// TwinCAT 3 PLC project Untitled1
// ProgramVersion: 3.1.0.9
// libraries:
//   Standard, * (System)
//   VisuElem3DPath, 3.5.6.0 (System)
//   VisuElemMeter, 3.5.6.0 (System)
//   VisuElems, 3.5.6.10 (System)
//   VisuElemsDateTime, 3.5.6.0 (System)
//   VisuElemsSpecialControls, 3.5.6.0 (System)
//   VisuElemsWinControls, 3.5.6.0 (System)
//   VisuElemTextEditor, 3.5.6.0 (System)
//   visuinputs, 3.5.6.0 (system)
//   VisuNativeControl, 3.5.6.0 (System)
//   Tc2_Standard, * (Beckhoff Automation GmbH)
//   Tc2_System, * (Beckhoff Automation GmbH)
//   Tc3_Interfaces, * (Beckhoff Automation GmbH)
//   Tc3_Module, * (Beckhoff Automation GmbH)
// project tree:
//   / GlobalTextList.TcGTLO, PlcTask.TcTTO, Visualization Manager.TcVMO (not stored)
//   POUs/ LADDER1.TcPOU, MAIN.TcPOU
//   VISUs/ Visualization.TcVIS
// real-time tasks:
//   TASK PlcTask: cycle T#10ms, priority 20, ADS port 350

CONFIGURATION Untitled1
    RESOURCE PLC ON TwinCAT3
        TASK PlcTask(INTERVAL := T#10ms, PRIORITY := 20);
        PROGRAM MAIN WITH PlcTask : MAIN;
    END_RESOURCE
END_CONFIGURATION

// ---- POUs/MAIN.TcPOU
PROGRAM MAIN
VAR
END_VAR

LADDER1();

END_PROGRAM

// ---- POUs/LADDER1.TcPOU
PROGRAM LADDER1
VAR
	stop: BOOL;
	start: BOOL;
	emergency: BOOL;
	S_place: BOOL;
	S_full: BOOL;
	S_empty: BOOL;
	S_loading: BOOL;
	S_unload: BOOL;
	valve: BOOL;
	Motor: BOOL;
	y1: BOOL;
	y3: BOOL;
	y2:BOOL;
	TankEmpty: BOOL;
    CU: BOOL; 
    RESET: BOOL; 
    PV: WORD; 
	FILLING: BOOL;
	CV: WORD;
	Q: Bool;
	counter: CTU;
END_VAR
VAR // added by the converter: edge detectors and wires of the graphical bodies
    _w1, _w2 : BOOL;
END_VAR

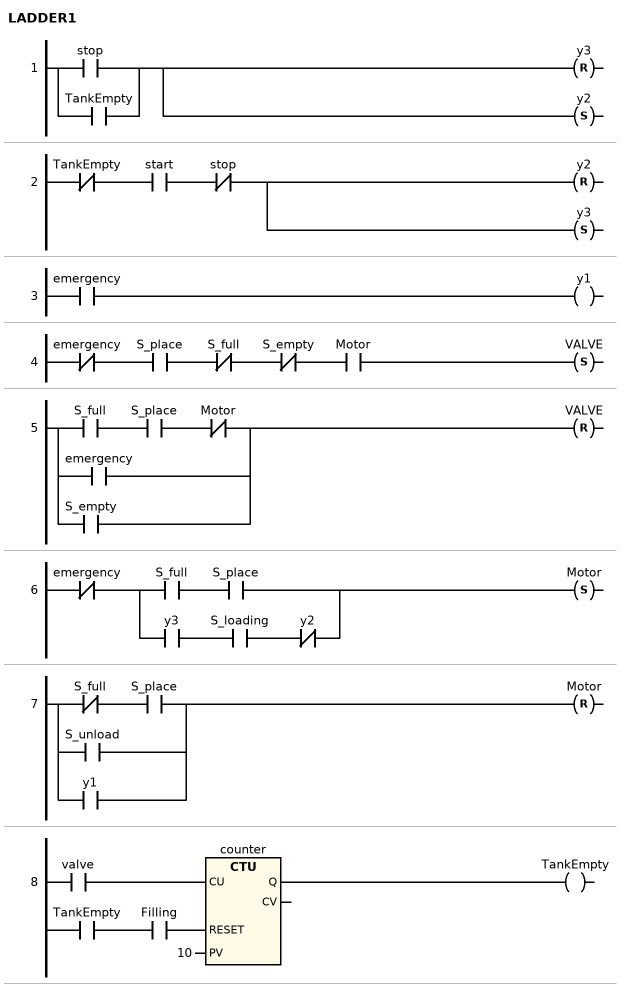
// NETWORK 1
_w1 := stop OR TankEmpty;
y3 R= _w1;
y2 S= _w1;

// NETWORK 2
_w2 := NOT TankEmpty AND start AND NOT stop;
y2 R= _w2;
y3 S= _w2;

// NETWORK 3
y1 := emergency;

// NETWORK 4
VALVE S= NOT emergency AND S_place AND NOT S_full AND NOT S_empty AND Motor;

// NETWORK 5
VALVE R= S_full AND S_place AND NOT Motor OR emergency OR S_empty;

// NETWORK 6
Motor S= NOT emergency AND (S_full AND S_place OR y3 AND S_loading AND NOT y2);

// NETWORK 7
Motor R= NOT S_full AND S_place OR S_unload OR y1;

// NETWORK 8
counter(CU := valve, RESET := TankEmpty AND Filling, PV := 10); // CTU
TankEmpty := counter.Q;

END_PROGRAM

// ---- GlobalTextList.TcGTLO
TEXTLIST GlobalTextList
  16 = 'CONTAINER FULL'
  17 = 'CONTAINER IN PLACE'
  22 = 'Counter : '
  23 = 'Counter : %d'
  24 = 'Counter : %i'
  21 = 'Counter : %s'
  2 = 'emergency'
  25 = 'Emergency Stop'
  26 = 'EMERGENCY STOP'
  13 = 'Filling'
  14 = 'LOADING'
  8 = 'Motor'
  18 = 'MOTOR'
  5 = 'S-empty'
  4 = 'S-full'
  6 = 'S-loading'
  3 = 'S-place'
  7 = 'S-unload'
  0 = 'start'
  1 = 'stop'
  11 = 'S_load'
  12 = 'S_loading'
  19 = 'TANK EMPTY'
  10 = 'tank-empty'
  15 = 'UNLOADING'
  9 = 'valve'
  20 = 'VALVE'
END_TEXTLIST

// ---- VISUs/Visualization.TcVIS
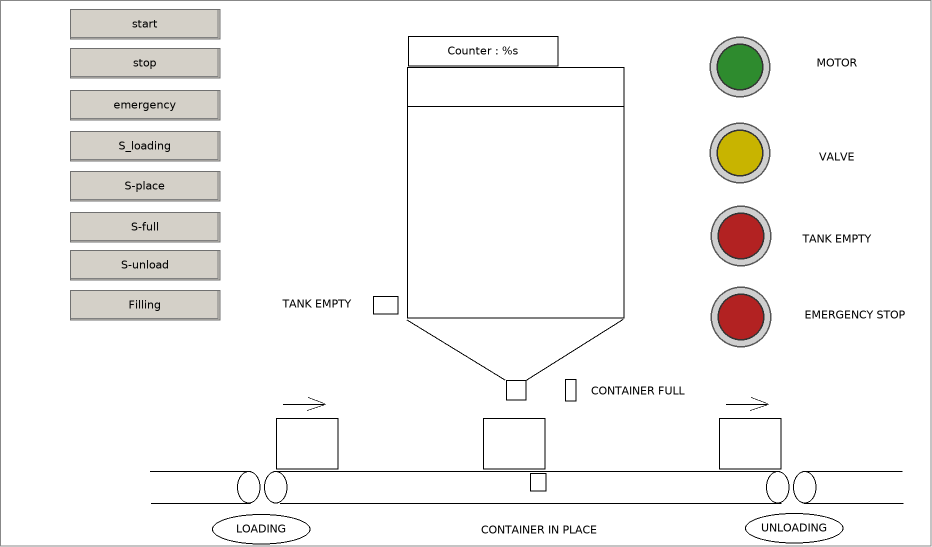
VISUALIZATION Visualization  // 932x547
    Lamp1 (705,32 70x70), variable: LADDER1.Motor, style: Lamp-Lamp1-Green
    Button (70,9 150x30), "start"
        OnMouseDown: toggle LADDER1.start
    Button (70,48 150x30), "stop"
        OnMouseDown: toggle LADDER1.stop
    Button (70,212 150x30), "S-full"
        OnMouseDown: toggle LADDER1.S_full
    Button (70,171 150x30), "S-place"
        OnMouseDown: toggle LADDER1.S_place
    Button (70,90 150x30), "emergency"
        OnMouseDown: toggle LADDER1.emergency
    Lamp1 (705,118 70x70), variable: LADDER1.valve, style: Lamp-Lamp1-Yellow
    Lamp1 (706,201 70x70), variable: LADDER1.TankEmpty, style: Lamp-Lamp1-Red
    Button (70,250 150x30), "S-unload"
        OnMouseDown: toggle LADDER1.S_unload
    Button (70,131 150x30), "S_loading"
        OnMouseDown: toggle LADDER1.S_loading
    Button (70,290 150x30), "Filling"
        OnMouseDown: toggle LADDER1.FILLING
    Rectangle (407,67 217x251)
    Rectangle (407,106 217x212), invisible if: LADDER1.TankEmpty
    Line (413,321)
    Line (505,380) (407,320)
    Line (585,354)
    Line (526,380) (623,319)
    Rectangle (506,380 20x20)
    Rectangle (483,418 62x51), colour toggle: LADDER1.S_full
        OnMouseDown: toggle LADDER1.S_full
    Rectangle (276,418 62x51)
    Rectangle (719,418 62x51)
    Line (726,404) (767,404)
    Line (751,397) (767,403)
    Line (750,410) (768,404)
    Line (283,404) (324,404)
    Line (308,397) (324,403)
    Line (307,410) (325,404)
    Ellipse (264,471 23x32)
    Line (278,471) (779,471)
    Ellipse (766,471 23x32)
    Line (280,503) (781,503)
    Ellipse (237,471 23x32)
    Ellipse (793,471 23x32)
    Line (803,471) (902,471)
    Line (804,503) (903,503)
    Line (150,471) (249,471)
    Line (151,503) (250,503)
    Ellipse (212,514 98x30), "LOADING"
    Ellipse (745,513 98x30), "UNLOADING"
    Rectangle (530,473 16x18)
    Rectangle (565,379 11x22)
    Label (549,376 178x30), "CONTAINER FULL"
    Label (464,515 150x30), "CONTAINER IN PLACE"
    Label (750,42 174x42), "MOTOR"
    Label (750,136 174x42), "VALVE"
    Label (750,218 174x42), "TANK EMPTY"
    Label (242,289 150x30), "TANK EMPTY"
    Rectangle (373,296 25x18)
    Rectangle (408,36 150x30), "Counter : %s", text variable: MAIN.LADDER1.counter.CV
    Lamp1 (706,282 70x70), variable: LADDER1.emergency, style: Lamp-Lamp1-Red
    Label (780,300 150x30), "EMERGENCY STOP"
END_VISUALIZATION
